Staubli VAL3: getValue_num.pgx

public program getValue_num(num& x_nValue[] (dimensions=1), string x_sItem (dimensions=1))
begin
  // Get IT
  if isDefined(cCount[x_sItem])
    x_nValue=cCount[x_sItem].nCount
  elseIf isDefined(aCount[x_sItem])
    x_nValue=aioGet(aCount[x_sItem].aAio)
  else
    // not found
    // toDO
    popUpMsg("value not found: "+x_sItem)
    x_nValue=-1
  endIf
end
